SUBAPPLICATION Uebung_011b1_AUDI (* Numeric Value Input ADD *)
  (* Standard: 61499-2; Description: Copyright (c) 2023 Meisterschulen am Ostbahnhof This program and the accompanying materials are made available under the terms of the Eclipse Public License 2.0 which is available at https://www.eclipse.org/legal/epl-2.0/ SPDX-License-Identifier: EPL-2.0 *)
  (* Version 1.0, 2026-04-14, Franz Höpfinger, Meisterschulen am Ostbahnhof, initial API and implementation and/or initial documentation *)
  PACKAGE Uebungen;
  IMPORT Uebungen::const::UT::DefaultPool::InputNumber_I1;
  IMPORT Uebungen::const::UT::DefaultPool::InputNumber_I2;
  IMPORT Uebungen::const::UT::DefaultPool::OutputNumber_N1;
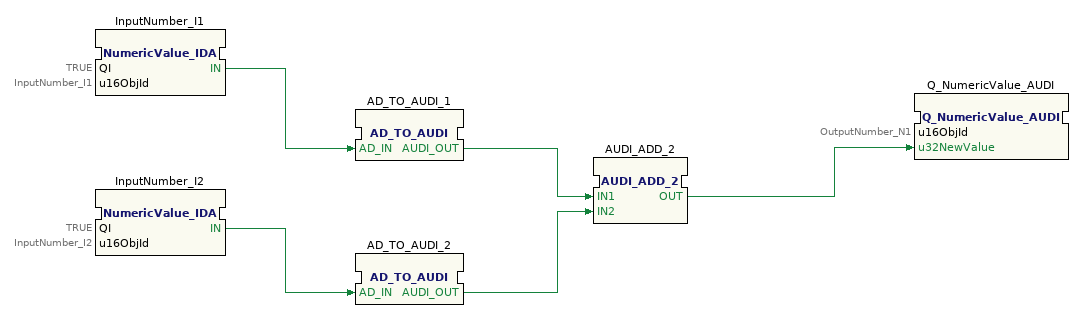
  FBS
    InputNumber_I1 : isobus::UT::io::NumericValue::NumericValue_IDA(QI := TRUE, u16ObjId := InputNumber_I1);
    InputNumber_I2 : isobus::UT::io::NumericValue::NumericValue_IDA(QI := TRUE, u16ObjId := InputNumber_I2);
    AD_TO_AUDI_1 : adapter::conversion::unidirectional::AD_TO_AUDI;
    AD_TO_AUDI_2 : adapter::conversion::unidirectional::AD_TO_AUDI;
    AUDI_ADD_2 : adapter::iec61131::arithmetic::AUDI_ADD_2;
    Q_NumericValue_AUDI : isobus::UT::Q::Q_NumericValue_AUDI(u16ObjId := OutputNumber_N1);
  END_FBS
  ADAPTER_CONNECTIONS
    InputNumber_I1.IN TO AD_TO_AUDI_1.AD_IN;
    InputNumber_I2.IN TO AD_TO_AUDI_2.AD_IN;
    AD_TO_AUDI_1.AUDI_OUT TO AUDI_ADD_2.IN1;
    AD_TO_AUDI_2.AUDI_OUT TO AUDI_ADD_2.IN2;
    AUDI_ADD_2.OUT TO Q_NumericValue_AUDI.u32NewValue;
  END_CONNECTIONS
END_SUBAPPLICATION
